FUNCTION_BLOCK FB_Zykluszeit
VAR_INPUT
	bStart:					BOOL;
	fZyklusZeitTask:		REAL;
END_VAR

VAR_OUTPUT
	fZyklusZeit:			REAL;
END_VAR

VAR
	fZykluszaehler:			REAL;
	fZykluszeitTemp:		REAL;
	fbStartFlanke:			R_TRIG;
	fbStopFlanke:			R_TRIG;
	bZyklusMessungAkt:		BOOL;
END_VAR

fbStartFlanke(CLK := bStart);
fbStopFlanke(CLK := NOT bStart);
fZykluszeitTemp := fZykluszaehler * (fZyklusZeitTask/1000);

IF fbStartFlanke.Q THEN
	fZykluszaehler := 0;
	fZyklusZeit := fZykluszeitTemp;
	bZyklusMessungAkt := FALSE;
END_IF

IF			fbStartFlanke.Q 
	AND NOT	bZyklusMessungAkt THEN
	bZyklusMessungAkt := TRUE;
END_IF

IF 		bZyklusMessungAkt THEN
	fZykluszaehler := fZykluszaehler + 1;
END_IF

IF			fbStopFlanke.Q 
	AND 	bZyklusMessungAkt THEN
	bZyklusMessungAkt := FALSE;
END_IF

(*
fbStartFlanke(CLK := bStart);
fbStopFlanke(CLK := bStop);
fZykluszeitTemp := fZykluszaehler * (fZyklusZeitTask/1000);

IF fbStartFlanke.Q THEN
	fZykluszaehler := 0;
	fZyklusZeit := fZykluszeitTemp;
	bZyklusMessungAkt := FALSE;
END_IF

IF			fbStartFlanke.Q 
	AND NOT	bZyklusMessungAkt THEN
	bZyklusMessungAkt := TRUE;
END_IF

IF 		bZyklusMessungAkt
	AND	MAIN.bProduzieren THEN
	fZykluszaehler := fZykluszaehler + 1;
END_IF

IF			fbStopFlanke.Q 
	AND 	bZyklusMessungAkt THEN
	bZyklusMessungAkt := FALSE;
END_IF
*)

END_FUNCTION_BLOCK

(* stored: Version 1.1.0.1, ProductVersion 3.1.4024.12
   POU FB_Zykluszeit: Id {725ba52a-6096-47c4-a78f-eda5b99a412c}, SpecialFunc None *)
